// Mitsubishi GX Works2 project: 240507_timechart12_ctr링카운터gxw   PLC: Q03UDV

PROGRAM MAIN
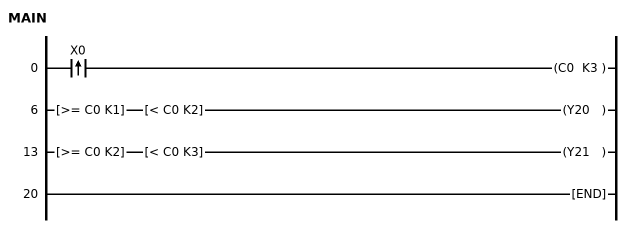
0     LDP     X0
      OUT     C0 K3
6     LD>=    C0 K1
      AND<    C0 K2
      OUT     Y20
13    LD>=    C0 K2
      AND<    C0 K3
      OUT     Y21
20    END
END_PROGRAM
